TYPE TcoTransferSystem_Status EXTENDS TcoCore.TcoStruct:
STRUCT


		ActionDescription:STRING;
		
END_STRUCT
END_TYPE

(* stored: Version 1.1.0.1
   DUT TcoTransferSystem_Status: Id {a17c8a6e-f30f-45cc-8e99-b971569c36c0} *)
